// TIA Portal V19 export
FUNCTION "Consumi" : Void   // FC51, LAD
// stored: SetENOAutomatically false
BEGIN

REGION Network 1: Lettura strumento PAC3220
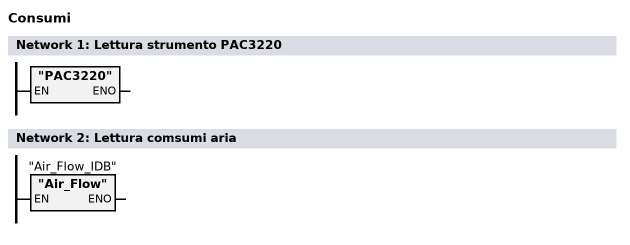
   RUNG wire#powerrail
      "PAC3220"()
   END_RUNG
   // the same network as SCL:
   "PAC3220"();
END_REGION

REGION Network 2: Lettura comsumi aria
   RUNG wire#powerrail
      "Air_Flow_IDB"()
   END_RUNG
   // the same network as SCL:
   "Air_Flow_IDB"();   // "Air_Flow"
END_REGION
END_FUNCTION
